# EPICS substitutions: evrSupport/Db/templates/autosave_evr.substitutions
#
# EVR autosave sample substitutions file
#
file autosave_evr.template
{
	{	IOC	= $(IOC),	EVR	= $(EVR)	}
}
